INTERFACE ITcoLogSink

METHOD Emit : BOOL
VAR_INPUT
	LogEvent		: REFERENCE TO LogEvent;
END_VAR
END_METHOD

END_INTERFACE

(* stored: Version 1.1.0.1, ProductVersion 3.1.4024.9
   Itf ITcoLogSink: Id {04cae3ff-198a-0a92-2922-2285610707ee}
   Method Emit: Id {2aa5cad7-93f9-03f1-260e-c3ea05c40b81} *)
